FUNCTION_BLOCK 
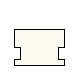
  EVENT_INPUT
    ;
  END_EVENT
  EVENT_OUTPUT
    ;
  END_EVENT
  VAR_INPUT
     : ;
     : ;
  END_VAR
  VAR_OUTPUT
     : ;
     : ;
     : ;
     : ;
  END_VAR
  ALGORITHM ALG IN ST:

  END_ALGORITHM
END_FUNCTION_BLOCK
(* other elements stored in the file *)
(* ECState name=START Initial=true *)
(* ECState name=BODY *)
(* ECAction Algorithm=ALG *)
(* ECTransition Source=START Destination=BODY *)
(* ECEventCondition Event=EP5 *)
(* ECTransition Source=BODY Destination=START_STATE *)
(* ECCondition  (LS <= LS1) *)
(* ECState Name=START_STATE *)
(* ECAction Output=START *)
